{attribute 'GeneratedUsingTerminal: ELX9410-0000-0018'}
{attribute addProperty BoxType "ELX9410-0000-0018"}
{attribute addProperty Description "ELX9410 E-Bus Power Supplier (Diagnostics)"}
{attribute addProperty Physics "KK"}
{attribute addProperty Id "Status_Us_InAT %I*Status_Us_In_B1E819A21Status_Us_OutAT %I*Status_Us_Out_B1E819A21WcStateAT %I*WcState_9091E0EB2InfoDataAT %I*InfoData_6F19DB2B2"}
{attribute addProperty CRC "144681044"}
{attribute addProperty Size "6"}
TYPE ELX9410_089FA854 EXTENDS EtcSlaveTerminalBase_947E5A46 :
STRUCT
	{attribute addProperty Name "Status_Us_In"}
	Status_Us_In : Status_Us_In_B1E819A2;
	{attribute addProperty Name "Status_Us_Out"}
	Status_Us_Out : Status_Us_Out_B1E819A2;
	{attribute addProperty Name "WcState"}
	WcState : WcState_9091E0EB;
	{attribute addProperty Name "InfoData"}
	InfoData : InfoData_6F19DB2B;
END_STRUCT
END_TYPE

(* stored: Version 1.2.0.0, ProductVersion 3.1.4024.9
   DUT ELX9410_089FA854: Id {b9c49f72-e432-4f18-b127-62d9b555818c} *)
